(* Logix 5000 project; controller Week_1_Intro_Studio_5000 Emulate 5570 rev 30.11; software revision 30.01 *)

TASK MainTask (continuous, watchdog 500 ms) : MainProgram
TASK tDecks (periodic, rate 10 ms, priority 10, watchdog 500 ms) : pInputs

MODULES
   Local : Emulate 5570 (ICP 2, rev 30.11)
END_MODULES

PROGRAM MainProgram   (* main routine MainRoutine *)

ROUTINE MainRoutine   (* ladder *)
END_ROUTINE

ROUTINE rInputsMain   (* ladder *)
END_ROUTINE
END_PROGRAM

PROGRAM pInputs   (* main routine rInputsMain *)

ROUTINE CelsiosToFahrenheit   (* ladder *)
END_ROUTINE

ROUTINE rInputsMain   (* ladder *)
END_ROUTINE

ROUTINE rMachineInputs   (* ladder *)
END_ROUTINE

ROUTINE rOpInput   (* ladder *)
END_ROUTINE

ROUTINE rPlcInputs   (* ladder *)
END_ROUTINE

ROUTINE rSmgInputs   (* ladder *)
END_ROUTINE
END_PROGRAM
